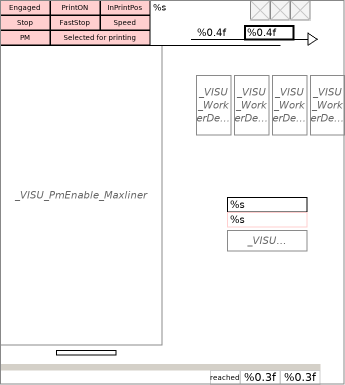
VISUALIZATION _VISU_Pm_Maxliner_mini_Worker  // 345x385
VAR_IN_OUT
  mInst : FB_PrintModule_Maxliner;
END_VAR
    Rectangle (150,0 160x15), "%s", text variable: mInst.fbAdsPm.stAds.aO_Name
    Rectangle (0,40 320x280)
    Frame (227,230 80x21)
        shows _VISU_MarkDetection_Trigger(mInst := mInst.fbMarkDetection)
    Rectangle (227,197 80x15), "%s", tooltip "active camera device", text variable: mInst.fbWorkerCamera._iActiveCam.sName
    Rectangle (227,212 80x15), "%s", tooltip "active camera mode", text variable: mInst.fbWorkerCamera._iActiveCam.eCameraMode, colour toggle: mInst.fbWorkerCamera._bCamValid
    RoundedRectangle (0,364 320x6), colour toggle: mInst.fbView.bMovingInd
    Frame (0,45 162x300)
        shows _VISU_PmEnable_Maxliner(mInst := mInst)
        p2738717112: mInst.fbView.zPos_PM
    RoundedRectangle (56,350 60x5), colour toggle: mInst.fbView.bPrintInd[1]
        p2738717112: mInst.fbView.zPos_PM
    Line (0,45) (280,45)
    RoundedRectangle (280,370 40x15), "%0.3f", tooltip "Target speed", text variable: mInst._pModuleMachineState^.fTargetSpeed
    RoundedRectangle (240,370 40x15), "%0.3f", tooltip "Current Speed", text variable: mInst.fSpeed
    RoundedRectangle (0,0 50x15), "Engaged", colour toggle: mInst._pModuleMachineState^.bEngaged
    RoundedRectangle (50,0 50x15), "PrintON", colour toggle: mInst._pModuleMachineState^.bPrintActivated
    RoundedRectangle (100,0 50x15), "InPrintPos", colour toggle: mInst._pModuleMachineState^.bUnitInPrintPosition
    RoundedRectangle (0,15 50x15), "Stop", colour toggle: NOT mInst._pModuleMachineState^.bStopRequest
    RoundedRectangle (50,15 50x15), "FastStop", colour toggle: NOT mInst._pModuleMachineState^.bFastStopRequest
    RoundedRectangle (100,15 50x15), "Speed", colour toggle: mInst.bSpeedReachedForPrinting
    Image (250,0 20x20), invisible if: NOT mInst._pModuleMachineState^.bSleep, image: ImagePool_Steinemann.sleep_icon
    Image (270,0 20x20), invisible if: NOT mInst._pModuleMachineState^.bShutdown, image: ImagePool_Steinemann.shutdown_icon
    Image (290,0 20x20), invisible if: NOT mInst._pModuleMachineState^.bEStop, image: ImagePool_Steinemann.estop_icon
    RoundedRectangle (210,370 30x15), "reached", tooltip "Target speed reached", colour toggle: mInst._pModuleMachineState^.bTargetSpeedReached
    Frame (234,75 35x60)
        shows _VISU_WorkerDefGrid_small(m_Inst := mInst.fbWorkerDeformation)
    Frame (272,75 35x60)
        shows _VISU_WorkerDefGrid_small(m_Inst := mInst.fbWorkerCamera)
    Frame (196,75 35x60)
        shows _VISU_WorkerDefGrid_small(m_Inst := mInst.fbWorkerPrint[1])
    RoundedRectangle (50,30 100x15), "Selected for printing"
        toggle mInst.bSelectedForPrint
    RoundedRectangle (0,30 50x15), "PM"
        toggle mInst.fbAdsPm.stAds.bI_Enable
    Rectangle (194,25 50x15), "%0.4f", tooltip "PM position on main tracker", text variable: mInst._fPmMainTrackPos
    Polyline (191,39) (308,39) (308,33) (317,39) (308,45) (308,39)
    Rectangle (244,25 50x15), "%0.4f", tooltip "PM position to previous", text variable: mInst._fPmDistToPrev
        OnMouseClick: write the text variable via Default
    Frame (310,75 35x60)
        shows _VISU_WorkerDefGrid_small(m_Inst := mInst.fbWorkerPython)
END_VISUALIZATION

(* stored: Version 1.1.0.1, ProductVersion 3.1.4024.11
   Visu _VISU_Pm_Maxliner_mini_Worker: Id {7b3f00dd-caff-4755-b0a0-9c29725d83aa} *)
